// TIA Portal V18 export
DATA_BLOCK "IR_Heater_Reduce_Peak"   // DB60
{ S7_Optimized_Access := 'TRUE' }
// stored: AutoNumber true, DBAccessibleFromOPCUA true, InstanceOfName IEC_TIMER, OfSystemLibElement IEC_TIMER, OfSystemLibVersion 1.0
"IEC_TIMER"
   // VAR
   //    PT : Time;
   //    ET { ExternalWritable := 'False'} : Time;
   //    IN : Bool;
   //    Q { ExternalWritable := 'False'} : Bool;
   // END_VAR
BEGIN
END_DATA_BLOCK
